{attribute addProperty BoxType "EK1122-0000-0018"}
{attribute addProperty Id "Beckhoff_EP4xxxsub_EK1100EK1100_179A0949162A_0001_EP4174_0002_0016EP4174_253CF8AE15219A_0002_EP4174_0002_0017EP4174_253CF8AE15219A_0003_EP4174_0002_0018EP4174_253CF8AE15219A_0004_EP4174_0002_0019EP4174_253CF8AE15219A_0005_EP4314_1002_0016EP4314_43F10CD122428A_0006_EP4374_0002_0016EP4374_55F3579519224A_0007_EP4374_0002_0017EP4374_D464211E19224A_0008_EP4374_0002_0018EP4374_D464211E19224A_0009_EP4374_0002_0019EP4374_D464211E19224A_0010_EP4378_1022_0017EP4378_6C133EE341652"}
{attribute addProperty CRC "623445774"}
{attribute addProperty SizeInBites "2032"}
{attribute addProperty SizeInBytes "254"}
TYPE Beckhoff_EP4xxxEK1122_2529070E EXTENDS EK1122_179A0949 :
STRUCT
	{attribute addProperty Name "Beckhoff_EP4xxxsub_EK1100"}
	Beckhoff_EP4xxxsub_EK1100 : EK1100_179A0949;
	{attribute addProperty Name "A_0001_EP4174_0002_0016"}
	A_0001_EP4174_0002_0016 : EP4174_253CF8AE;
	{attribute addProperty Name "A_0002_EP4174_0002_0017"}
	A_0002_EP4174_0002_0017 : EP4174_253CF8AE;
	{attribute addProperty Name "A_0003_EP4174_0002_0018"}
	A_0003_EP4174_0002_0018 : EP4174_253CF8AE;
	{attribute addProperty Name "A_0004_EP4174_0002_0019"}
	A_0004_EP4174_0002_0019 : EP4174_253CF8AE;
	{attribute addProperty Name "A_0005_EP4314_1002_0016"}
	A_0005_EP4314_1002_0016 : EP4314_43F10CD1;
	{attribute addProperty Name "A_0006_EP4374_0002_0016"}
	A_0006_EP4374_0002_0016 : EP4374_55F35795;
	{attribute addProperty Name "A_0007_EP4374_0002_0017"}
	A_0007_EP4374_0002_0017 : EP4374_D464211E;
	{attribute addProperty Name "A_0008_EP4374_0002_0018"}
	A_0008_EP4374_0002_0018 : EP4374_D464211E;
	{attribute addProperty Name "A_0009_EP4374_0002_0019"}
	A_0009_EP4374_0002_0019 : EP4374_D464211E;
	{attribute addProperty Name "A_0010_EP4378_1022_0017"}
	A_0010_EP4378_1022_0017 : EP4378_6C133EE3;
END_STRUCT
END_TYPE

(* stored: Version 1.2.0.0, ProductVersion 3.1.4024.9
   DUT Beckhoff_EP4xxxEK1122_2529070E: Id {39124629-bcd7-4a4a-afe6-ce422e633a62} *)
